FUNCTION_BLOCK FB_MSSQL_spUpdateBatchToProductionQueue
VAR_INPUT
	Execute					: BOOL;
	Enable					: BOOL;
	Reset					: BOOL;
	BatchId	: STRING(DB.MAX_STRING_SIZE);
	BatchInfoJson	: STRING(DB.MAX_STRING_SIZE);
	BatchItemsJson	: STRING(DB.MAX_STRING_SIZE);
END_VAR
VAR_OUTPUT
	Error					: BOOL;
	ErrorID					: DINT;
	Done					: BOOL;
	Busy					: BOOL;
	tcMessage 				: I_TcMessage;
	Q_tElapsedTime			: TIME;
END_VAR
VAR
	RTRIG_Execute			: R_TRIG;
	RTRIG_Reset				: R_TRIG;
	iState					: INT := -1;
	TON_Read				: TON;
	Parameters				: DUT_stUpdateBatchToProductionQueue;
END_VAR
VAR_IN_OUT
	fbSQLResult				: FB_SQLResultEvt;
	fbSQLStoredProcedure	: FB_SQLStoredProcedureEvt;
END_VAR

RTRIG_Reset(CLK := Reset);
IF RTRIG_Reset.Q AND Execute AND Error AND NOT Busy THEN
	Execute := FALSE;
END_IF

Parameters.BatchId := BatchId;
Parameters.BatchInfoJson := BatchInfoJson;
Parameters.BatchItemsJson := BatchItemsJson;
RTRIG_Execute(CLK := Execute AND Enable);
IF(RTRIG_Execute.Q) THEN
	 Done							:= FALSE;
	 Error							:= FALSE;
	 ErrorID						:= 0;
	 
	 iState							:= 0;
ELSIF NOT Execute AND NOT Busy THEN
	Busy			:= FALSE;
	Done			:= FALSE;
	Error			:= FALSE;
	
	iState := -1;
END_IF
 
 // Elapsed Time
 TON_Read(PT:= T#5S);
 
 CASE iState OF
 
	 0:
	 		TON_Read.IN 						:= FALSE;
			Busy								:= TRUE;
			iState 								:= 10;
		
	10:
		IF fbSQLStoredProcedure.Execute(pParameterStrc := ADR(Parameters), cbParameterStrc:= SIZEOF(Parameters)) THEN
			TON_Read.IN := TRUE;
			IF fbSQLStoredProcedure.bError THEN
				tcMessage := fbSQLStoredProcedure.ipTcResult;
				
				iState 							:= 1010;
			ELSE
				iState 							:= 999;
			END_IF    
		END_IF
		
//	20:
//		iState 							:= 999;
//		IF fbSQLResult.Read(0, fbSQLResult.nDataCount, ADR(Result), SIZEOF(Result), FALSE, TRUE) THEN
//			IF fbSQLResult.bError THEN
//				iState 							:= 1020;
//			ELSE
				
//				iState 							:= 30;
//			END_IF
//		END_IF
		
//	30: 
//		IF fbSQLResult.Release() THEN
//			iState 								:= 999;	
//		END_IF
		
	999:
		TON_Read.IN 	:= FALSE;
		Done			:= TRUE;
		Busy			:= FALSE;
		
 END_CASE 
 
IF iState > 1000 THEN
	Error 		:= TRUE;
	ErrorID	 	:= iState;
	Busy	 	:= FALSE;
	TON_Read.IN := FALSE;
	iState := -1;
END_IF

END_FUNCTION_BLOCK

(* stored: Version 1.1.0.1, ProductVersion 3.1.4024.15
   POU FB_MSSQL_spUpdateBatchToProductionQueue: Id {5c2b3f54-f13c-40ad-b993-b6565621072b}, SpecialFunc None *)
